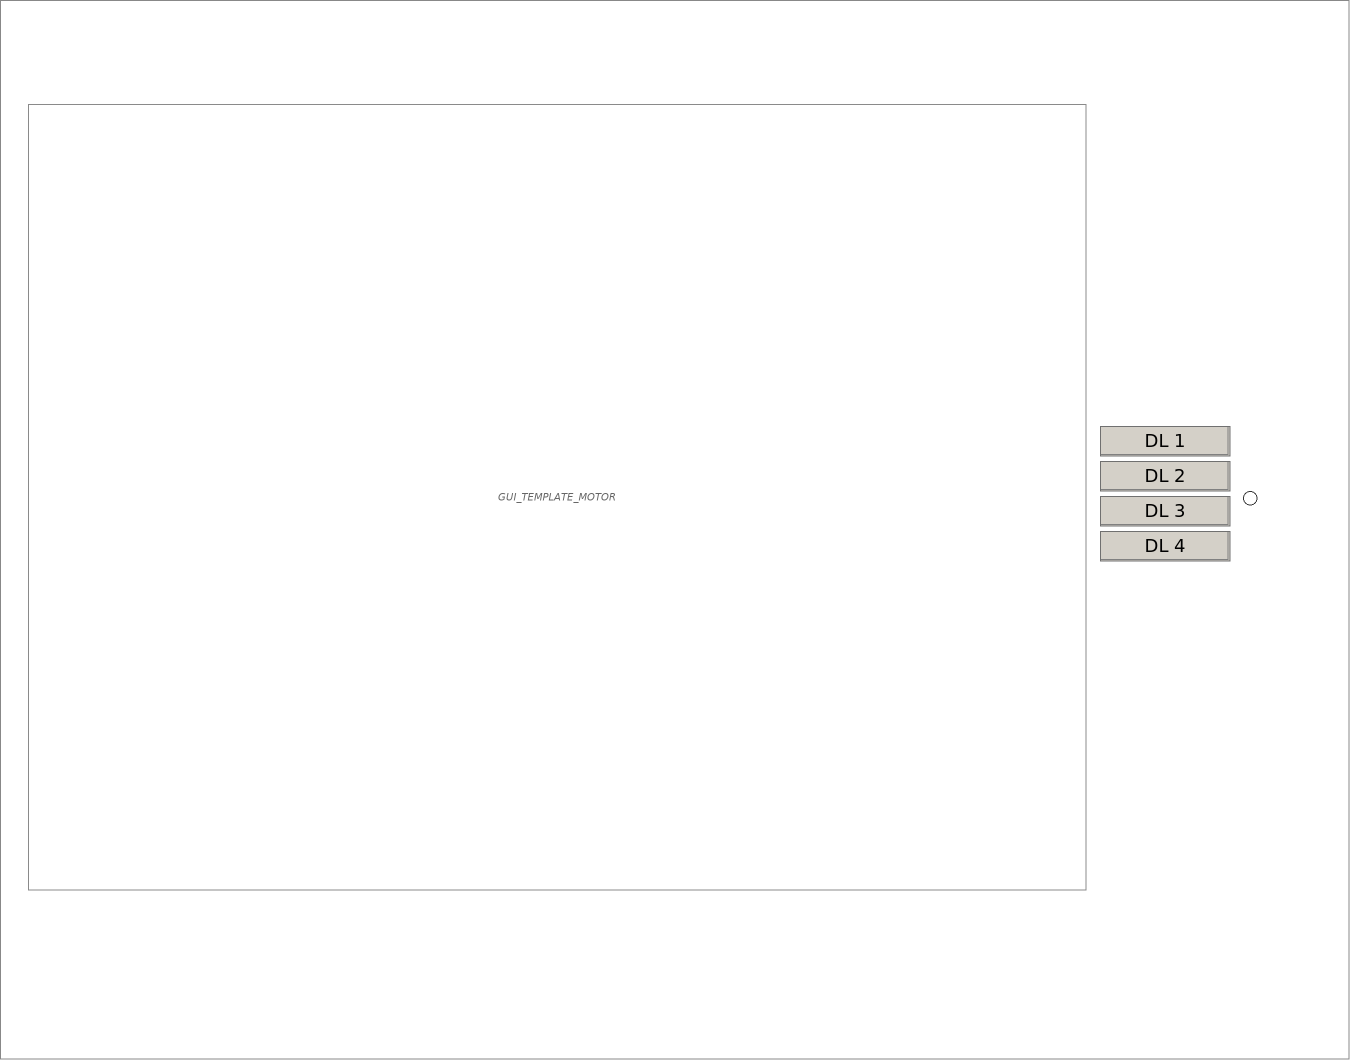
VISUALIZATION VISU_HMI_DELAY_LINES  // 1350x1060
    Label (10,10 199x30), "Delay Lines"
    Group (28,104 1260x786)
        Frame (0,0 1058x786)
            shows GUI_TEMPLATE_MOTOR(m_Instance := MAIN.nott_ics.Delay_Lines.ptrDelayLines[MAIN.nott_ics.Delay_Lines.guiShutterIndex]^)
        Group (1072,322 188x142)
            RadioButton (141,2 47x140), variable: MAIN.nott_ics.Delay_Lines.guiShutterIndex-1
                Areas[0]: Text=Radiobutton
                Areas[1]: Text=Radiobutton
            Button (0,0 130x30), "DL 1"
                OnMouseClick: execute { MAIN.nott_ics.Delay_Lines.guiShutterIndex := 1; }
            Button (0,35 130x30), "DL 2"
                OnMouseClick: execute { MAIN.nott_ics.Delay_Lines.guiShutterIndex := 2; }
            Button (0,70 130x30), "DL 3"
                OnMouseClick: execute { MAIN.nott_ics.Delay_Lines.guiShutterIndex := 3; }
            Button (0,105 130x30), "DL 4"
                OnMouseClick: execute { MAIN.nott_ics.Delay_Lines.guiShutterIndex := 4; }
END_VISUALIZATION

(* stored: Version 1.1.0.1, ProductVersion 3.1.4024.14
   Visu VISU_HMI_DELAY_LINES: Id {a7164e6a-3907-4853-957e-398d9bd38f26} *)
